Omron CX-Programmer project NewProject (CX-Programmer 9.03)

# PLC APK46: CS1H CPU63
; KARTONIKARKA

## Program TASK_MENAGER (cyclic task 0)
Local symbols
AWARIA_ZBIORCZA 49.15 BOOL  ; AWARIA ZBIORCZA KARTONIKARKI
A_21_22_A1 0.10 BOOL  ; TRIP-NAPĘDÓW
A_21_28 2.04 BOOL  ; ODBLOKOWANIE NAPĘDU GŁÓWNEGO
A_21_A2 0.11 BOOL  ; NAPĘD GŁÓWNY PO BAZOWANIU
A_21_E1 2.05 BOOL  ; JOG-NAPĘDU GŁÓWNEGO
A_21_E2 2.06 BOOL  ; PROGRAM START- TRIP NAPĘDU GŁÓWNEGO
A_21_E3 2.07 BOOL  ; BAZOWANIE NAPĘDU GŁÓWNEGO
A_21_E4 2.08 BOOL  ; INICJACJA NAPĘDU GŁÓWNEGO
A_21_E5 2.09 BOOL  ; input 5 napędu głównego
A_22_28 2.10 BOOL  ; ODBLOKOWANIE NAPĘlDU ZAMYKANIA
A_22_A2 0.12 BOOL  ; NAPĘDU ZAKLEJANIA KARTONIKÓW PO BAZOWANIU
A_22_E1 2.11 BOOL  ; PROGRAM START NAPĘDU ZAMYANA
A_22_E2 2.12 BOOL  ; BAZOWANE NAPĘDU ZAMYKANIA
A_22_E3 2.13 BOOL  ; NCJACJA NAPĘDU ZAMYKANIA
A_22_E4 2.14 BOOL
A_22_E5 2.15 BOOL
CAM_1 25.00 BOOL  ; ZATRZYMANIE SILNIKA
GOT_KART 201.00 BOOL  ; GOTOWOŚĆ KARTONIKARKI DO PRZYJĘCIA PRODUKTU
GOT_KLEJU 0.13 BOOL  ; GOTOWOŚĆ KLEJARKI NORDSON
K_131 2.00 BOOL  ; STYCZNIK-NAPĘD GŁÓWNY
K_132 2.01 BOOL  ; STYCZNIK TRANSPORTER
K_133 2.02 BOOL  ; STYCZNIK KLEJARKA
K_168 3.15 BOOL  ; PRZEKAŻNIK DRUKARKI
K_174 3.11 BOOL  ; PRZEKAŻNIK GOTOWOŚĆ
K_175 3.12 BOOL  ; PRZEKAŻNIK AWARIA
OBW_BEZPIECZ 0.14 BOOL  ; OBWÓD BEZPIECZEŃSTWA
OBW_OSŁON 0.15 BOOL  ; OBWÓD  OSŁON
OBW_STOP 0.14 BOOL  ; OBWÓD STOP
OBW_STOP_OSŁON 0.15 BOOL  ; OBWÓD STOPU I OSŁON
POZ_1024_0 0.00 BOOL  ; BIT 0 ENCODERA
POZ_1024_1 0.01 BOOL  ; BIT 1 ENCODERA
POZ_1024_2 0.02 BOOL  ; BIT 2 ENCODERA
POZ_1024_3 0.03 BOOL  ; BIT 3 ENCODERA
POZ_1024_4 0.04 BOOL  ; BIT 4 ENCODERA
POZ_1024_5 0.05 BOOL  ; BIT 5 ENCODERA
POZ_1024_6 0.06 BOOL  ; BIT 6 ENCODERA
POZ_1024_7 0.07 BOOL  ; BIT 7 ENCODERA
POZ_1024_8 0.08 BOOL  ; BIT 8 ENCODERA
POZ_1024_9 0.09 BOOL  ; BIT 9 ENCODERA
Q_32 1.00 BOOL  ; ZABEZPIECZENIE TERMICZNE TRANSPORTERA
REZERWA_OUT 2.03 BOOL
Restart_specjal_IO A502.00 BOOL
Run_DP 2000.00 BOOL
START W2.00 BOOL  ; ZAŁĄCZONA MASZYNA DO PRACY
S_111L 3.10 BOOL  ; LAMPKA ZAŁĄCZENIE
S_112 1.01 BOOL  ; PRZYCISK ZAŁĄCZENIE
S_113 1.02 BOOL  ; PRZYCISK W YŁĄCZENIE
S_114 1.03 BOOL  ; FOTOKOMÓRKA OBECNOŚCI PAKIETU NA TRANSPORTERZE
S_115 1.04 BOOL  ; OBECNOŚĆ PAKIETU NAD PODNOSZENIEM
S_116 1.05 BOOL  ; FOTOKOMÓRKA OBECNOŚCI KARTONIKA
S_117 1.06 BOOL  ; CZUJNIKI POZYCJI ZAKLEJANIA KARTONIKA
S_118 1.07 BOOL  ; PODNIESIENIE PAKIETU POCZĄTEK
S_121 1.08 BOOL  ; KONIEC SIŁOWNIKA PODNOSZĄCEGO PAKIET
S_122 1.09 BOOL  ; POCZĄTEK SIŁOWNIKA KLAPEK BOCZNYCH
S_123 1.10 BOOL  ; KONIEC SIŁOWNIKA KLAPEK BOCZNYCH
S_124 1.11 BOOL  ; POCZĄTEK SIŁOWNIKA POBIERAJĄCEGO KARTONIK
S_125 1.12 BOOL  ; KONIEC  SIŁOWNIKA POBIERAJĄCEGO KARTONIK
S_126 1.13 BOOL  ; POCZĄTEK SIŁOWNIKA WPYCHAJĄCEGO PAKIET
S_127 1.14 BOOL  ; KONIEC SIŁOWNIKA WPYCHAJĄCEGO
S_128 1.15 BOOL  ; FOTOKOMÓRKA WYJKRYWAJĄCA KARTONIK PRZED SKLEJENIEM
Y_151 3.00 BOOL  ; POBIERANIE KARTONIKÓW
Y_152 3.01 BOOL  ; EŻEKTOR
Y_153 3.02 BOOL  ; PODNOSZENIE PAKIETU
Y_154 3.03 BOOL  ; WPYCHANIE PAKIETU
Y_155 3.04 BOOL  ; KLAPKI BOCZNE
Y_156 3.05 BOOL  ; TRANSPORTER NA STOJAKU
Y_157 3.06 BOOL  ; SPUST POWIETRZA
Y_161 3.08 BOOL  ; ZAWÓR APLIKACJI KLEJU 1
Y_162 3.09 BOOL  ; ZAWÓR APLIKACJI KLEJU 2
ZAŁĄCZ_SILNIKI W0.01 BOOL  ; ZAŁĄCZONE SILNIKI
ZAŁĄCZ_STER W0.00 BOOL  ; ZAŁĄCZONE STEROWANIE
cam_1 25.00 BOOL  ; zatrzymanie napędu głównego
cam_10 25.09 BOOL
cam_2 25.01 BOOL
cam_3 25.02 BOOL
cam_4 25.03 BOOL
cam_5 25.04 BOOL
cam_6 25.05 BOOL
cam_7 25.06 BOOL
cam_8 25.07 BOOL
cam_9 25.08 BOOL

### Section inicjacja

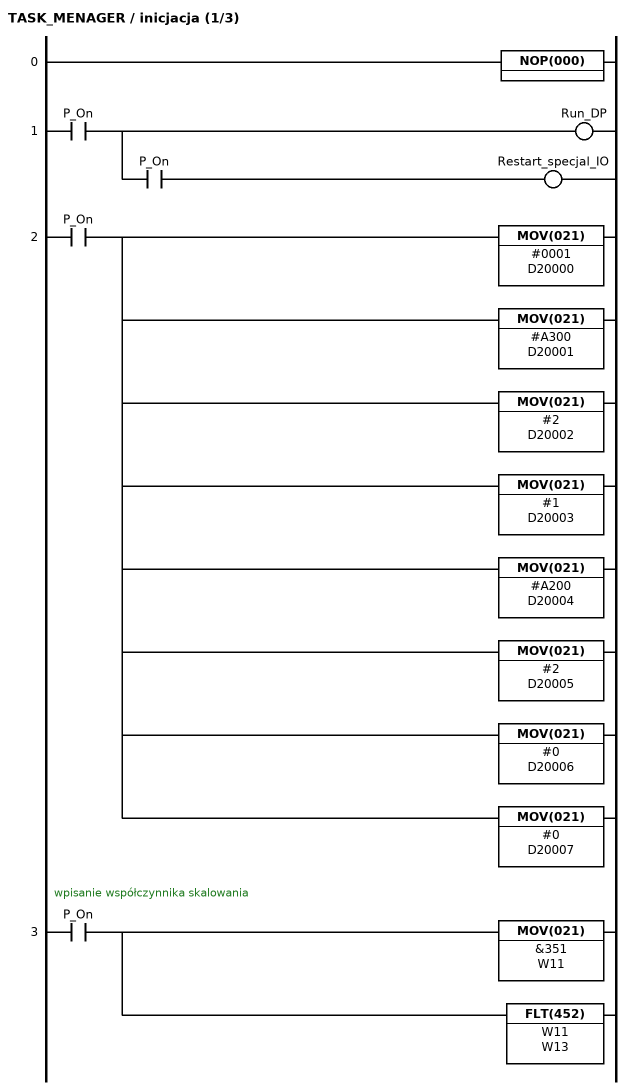
; rung 0
NOP(000)
; rung 1
LD P_On
OUT Run_DP
AND P_On
OUT Restart_specjal_IO
; rung 2
LD P_On
MOV(021) #0001 D20000  // jeden obszar wyjściowy
MOV(021) #A300 D20001  // początek obszaru wyjściowego
MOV(021) #2 D20002  // ustawienie 4 słów wejściowych
MOV(021) #1 D20003  // ustawienie jednego obszaru wyjsciowego
MOV(021) #A200 D20004  // początek obszaru wejściowego
MOV(021) #2 D20005  // ustawienie 4 słów wyjściowych
MOV(021) #0 D20006
MOV(021) #0 D20007
; rung 3: wpisanie współczynnika skalowania
LD P_On
MOV(021) &351 W11
FLT(452) W11 W13

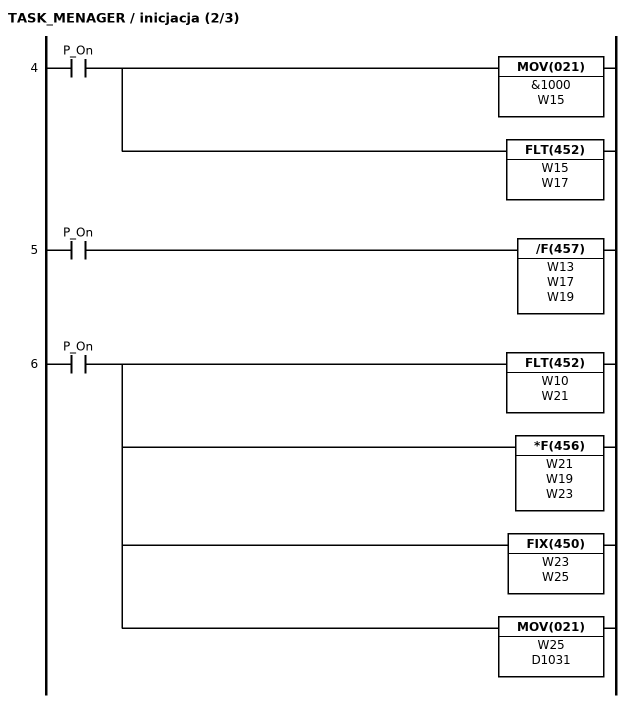
; rung 4
LD P_On
MOV(021) &1000 W15
FLT(452) W15 W17
; rung 5
LD P_On
/F(457) W13 W17 W19  // wspolczynnik 0,351
; rung 6
LD P_On
FLT(452) W10 W21
*F(456) W21 W19 W23
FIX(450) W23 W25
MOV(021) W25 D1031

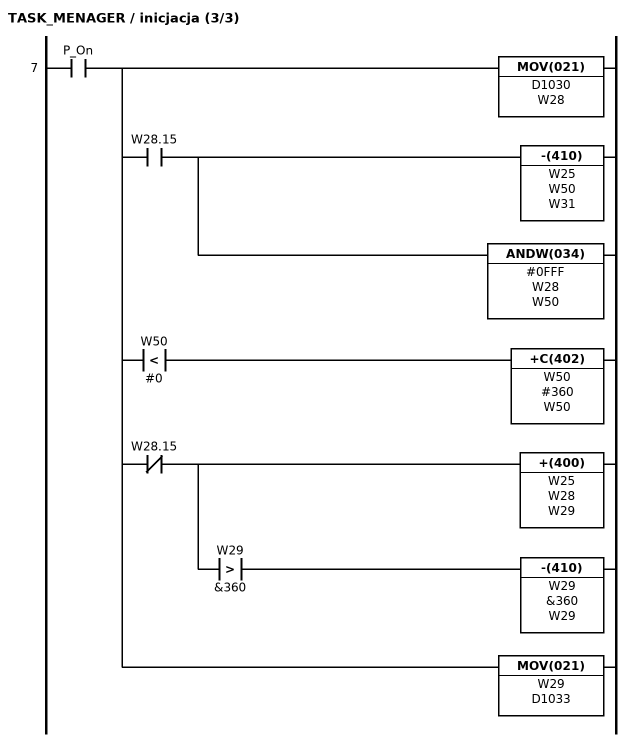
; rung 7
LD P_On
OUT TR0
MOV(021) D1030 W28
AND W28.15
-(410) W25 W50 W31
ANDW(034) #0FFF W28 W50
LD TR0
AND<S(312) W50 #0
+C(402) W50 #360 W50
LD TR0
ANDNOT W28.15
+(400) W25 W28 W29
AND>(320) W29 &360
-(410) W29 &360 W29
LD TR0
MOV(021) W29 D1033

### Section cam_section

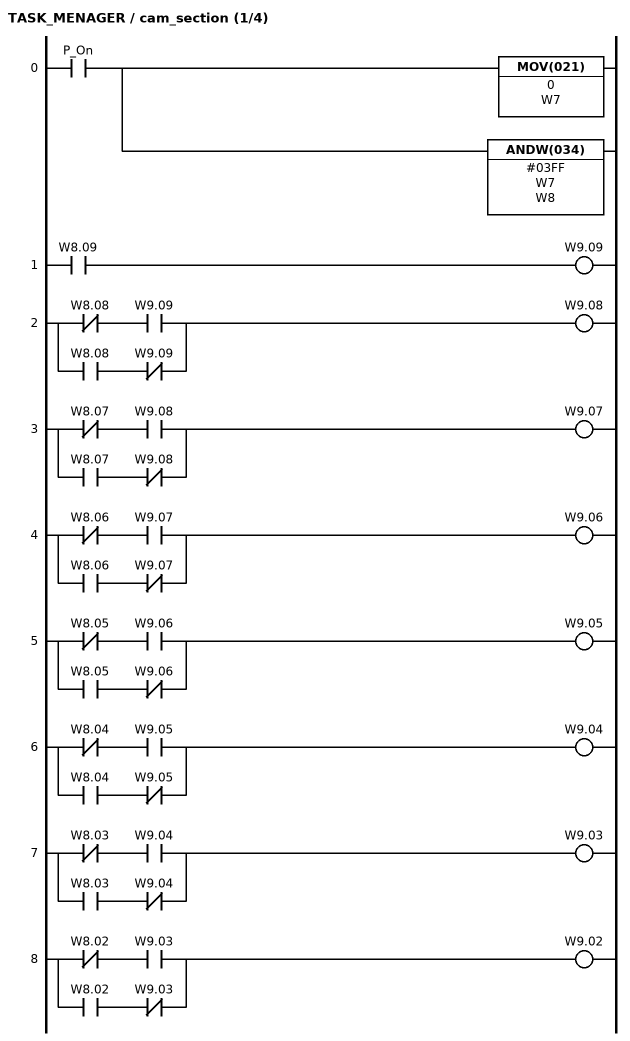
; rung 0
LD P_On
MOV(021) 0 W7
ANDW(034) #03FF W7 W8
; rung 1
LD W8.09
OUT W9.09
; rung 2
LDNOT W8.08
AND W9.09
LD W8.08
ANDNOT W9.09
ORLD
OUT W9.08
; rung 3
LDNOT W8.07
AND W9.08
LD W8.07
ANDNOT W9.08
ORLD
OUT W9.07
; rung 4
LDNOT W8.06
AND W9.07
LD W8.06
ANDNOT W9.07
ORLD
OUT W9.06
; rung 5
LDNOT W8.05
AND W9.06
LD W8.05
ANDNOT W9.06
ORLD
OUT W9.05
; rung 6
LDNOT W8.04
AND W9.05
LD W8.04
ANDNOT W9.05
ORLD
OUT W9.04
; rung 7
LDNOT W8.03
AND W9.04
LD W8.03
ANDNOT W9.04
ORLD
OUT W9.03
; rung 8
LDNOT W8.02
AND W9.03
LD W8.02
ANDNOT W9.03
ORLD
OUT W9.02

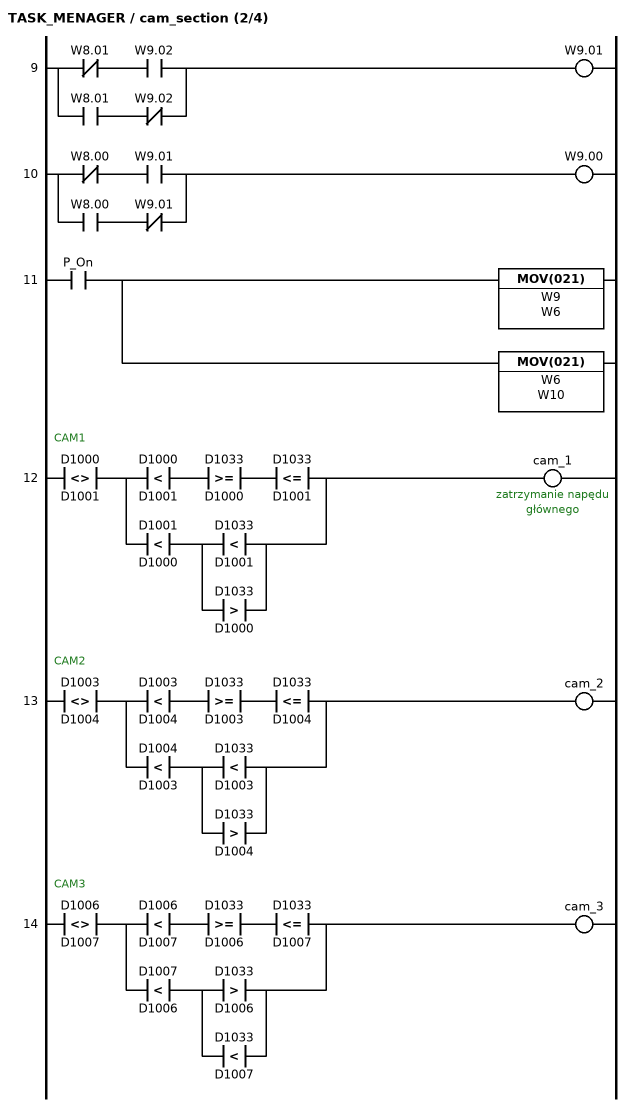
; rung 9
LDNOT W8.01
AND W9.02
LD W8.01
ANDNOT W9.02
ORLD
OUT W9.01
; rung 10
LDNOT W8.00
AND W9.01
LD W8.00
ANDNOT W9.01
ORLD
OUT W9.00
; rung 11
LD P_On
MOV(021) W9 W6
MOV(021) W6 W10
; rung 12: CAM1
LD<>(305) D1000 D1001
LD<(310) D1000 D1001
AND>=(325) D1033 D1000
AND<=(315) D1033 D1001
LD<(310) D1001 D1000
LD<(310) D1033 D1001
OR>(320) D1033 D1000
ANDLD
ORLD
ANDLD
OUT cam_1  ; zatrzymanie napędu głównego
; rung 13: CAM2
LD<>(305) D1003 D1004
LD<(310) D1003 D1004
AND>=(325) D1033 D1003
AND<=(315) D1033 D1004
LD<(310) D1004 D1003
LD<(310) D1033 D1003
OR>(320) D1033 D1004
ANDLD
ORLD
ANDLD
OUT cam_2
; rung 14: CAM3
LD<>(305) D1006 D1007
LD<(310) D1006 D1007
AND>=(325) D1033 D1006
AND<=(315) D1033 D1007
LD<(310) D1007 D1006
LD>(320) D1033 D1006
OR<(310) D1033 D1007
ANDLD
ORLD
ANDLD
OUT cam_3

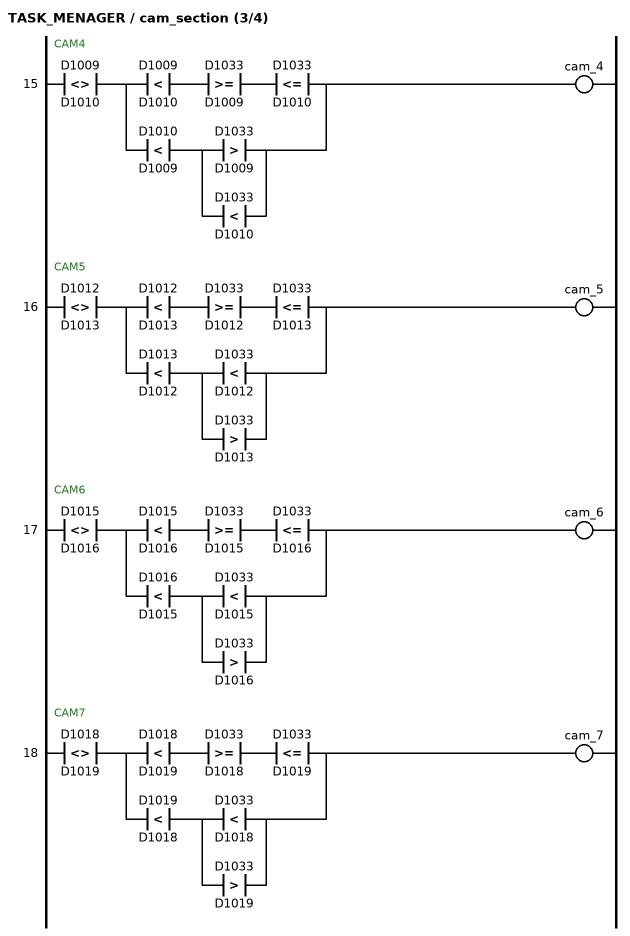
; rung 15: CAM4
LD<>(305) D1009 D1010
LD<(310) D1009 D1010
AND>=(325) D1033 D1009
AND<=(315) D1033 D1010
LD<(310) D1010 D1009
LD>(320) D1033 D1009
OR<(310) D1033 D1010
ANDLD
ORLD
ANDLD
OUT cam_4
; rung 16: CAM5
LD<>(305) D1012 D1013
LD<(310) D1012 D1013
AND>=(325) D1033 D1012
AND<=(315) D1033 D1013
LD<(310) D1013 D1012
LD<(310) D1033 D1012
OR>(320) D1033 D1013
ANDLD
ORLD
ANDLD
OUT cam_5
; rung 17: CAM6
LD<>(305) D1015 D1016
LD<(310) D1015 D1016
AND>=(325) D1033 D1015
AND<=(315) D1033 D1016
LD<(310) D1016 D1015
LD<(310) D1033 D1015
OR>(320) D1033 D1016
ANDLD
ORLD
ANDLD
OUT cam_6
; rung 18: CAM7
LD<>(305) D1018 D1019
LD<(310) D1018 D1019
AND>=(325) D1033 D1018
AND<=(315) D1033 D1019
LD<(310) D1019 D1018
LD<(310) D1033 D1018
OR>(320) D1033 D1019
ANDLD
ORLD
ANDLD
OUT cam_7

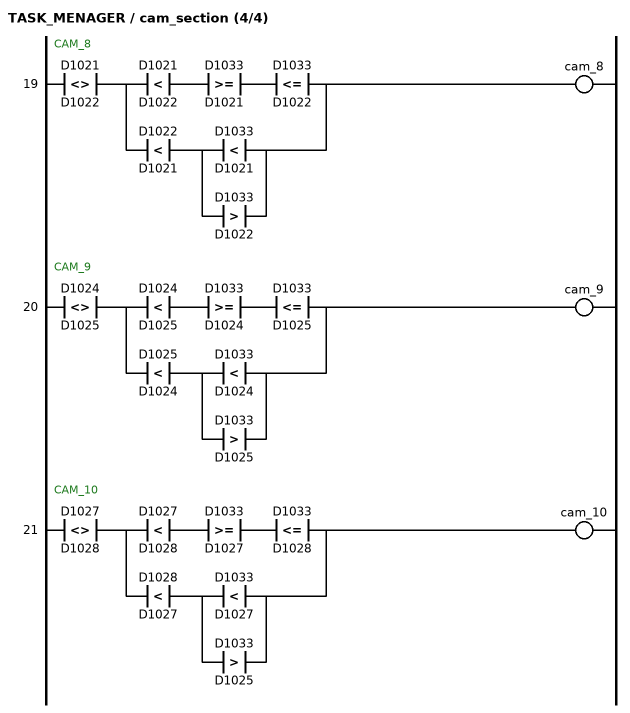
; rung 19: CAM_8
LD<>(305) D1021 D1022
LD<(310) D1021 D1022
AND>=(325) D1033 D1021
AND<=(315) D1033 D1022
LD<(310) D1022 D1021
LD<(310) D1033 D1021
OR>(320) D1033 D1022
ANDLD
ORLD
ANDLD
OUT cam_8
; rung 20: CAM_9
LD<>(305) D1024 D1025
LD<(310) D1024 D1025
AND>=(325) D1033 D1024
AND<=(315) D1033 D1025
LD<(310) D1025 D1024
LD<(310) D1033 D1024
OR>(320) D1033 D1025
ANDLD
ORLD
ANDLD
OUT cam_9
; rung 21: CAM_10
LD<>(305) D1027 D1028
LD<(310) D1027 D1028
AND>=(325) D1033 D1027
AND<=(315) D1033 D1028
LD<(310) D1028 D1027
LD<(310) D1033 D1027
OR>(320) D1033 D1025
ANDLD
ORLD
ANDLD
OUT cam_10

### Section przyjęcie_pakietu

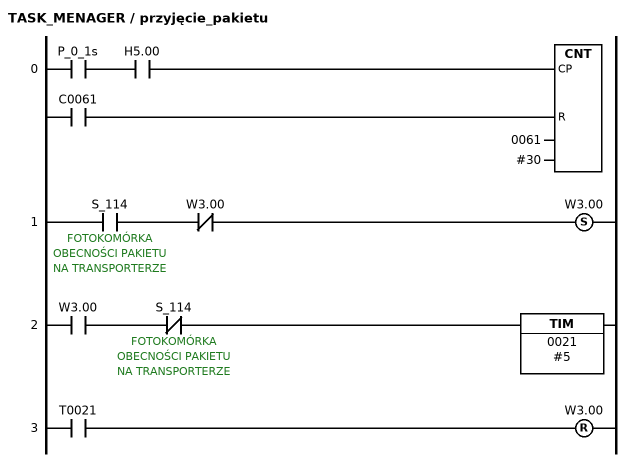
; rung 0
LD P_0_1s
AND H5.00
LD C0061
CNT 0061 #30
; rung 1
LD S_114  ; FOTOKOMÓRKA OBECNOŚCI PAKIETU NA TRANSPORTERZE
ANDNOT W3.00
SET W3.00
; rung 2
LD W3.00
ANDNOT S_114  ; FOTOKOMÓRKA OBECNOŚCI PAKIETU NA TRANSPORTERZE
TIM 0021 #5
; rung 3
LD T0021
RSET W3.00

### Section awaria

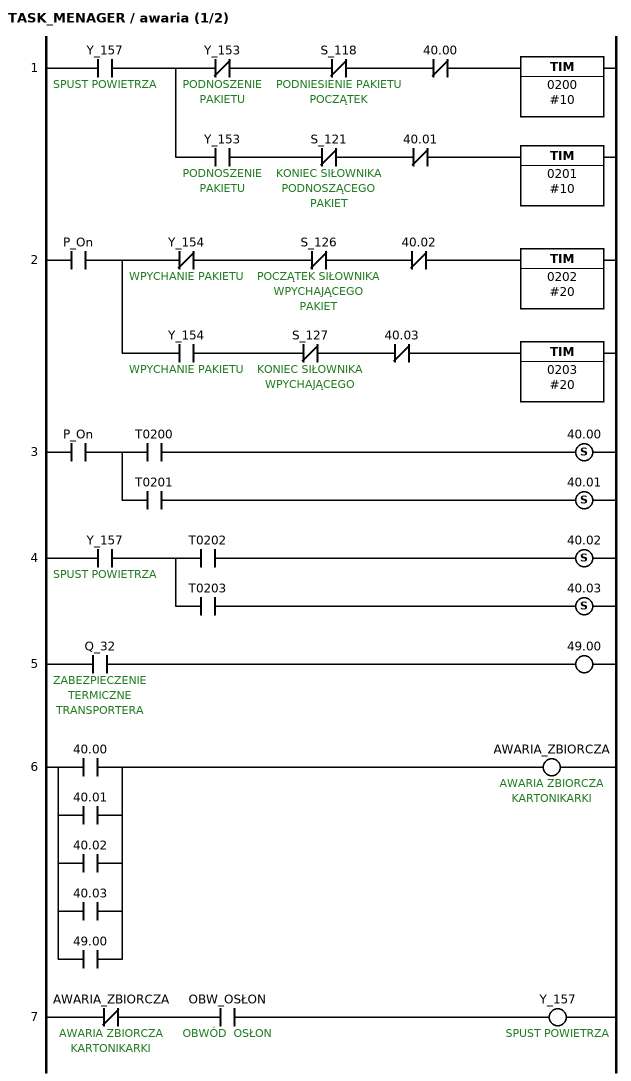
; rung 1
LD Y_157  ; SPUST POWIETRZA
OUT TR0
ANDNOT Y_153  ; PODNOSZENIE PAKIETU
ANDNOT S_118  ; PODNIESIENIE PAKIETU POCZĄTEK
ANDNOT 40.00
TIM 0200 #10
LD TR0
AND Y_153  ; PODNOSZENIE PAKIETU
ANDNOT S_121  ; KONIEC SIŁOWNIKA PODNOSZĄCEGO PAKIET
ANDNOT 40.01
TIM 0201 #10
; rung 2
LD P_On
OUT TR0
ANDNOT Y_154  ; WPYCHANIE PAKIETU
ANDNOT S_126  ; POCZĄTEK SIŁOWNIKA WPYCHAJĄCEGO PAKIET
ANDNOT 40.02
TIM 0202 #20
LD TR0
AND Y_154  ; WPYCHANIE PAKIETU
ANDNOT S_127  ; KONIEC SIŁOWNIKA WPYCHAJĄCEGO
ANDNOT 40.03
TIM 0203 #20
; rung 3
LD P_On
OUT TR0
AND T0200
SET 40.00
LD TR0
AND T0201
SET 40.01
; rung 4
LD Y_157  ; SPUST POWIETRZA
OUT TR0
AND T0202
SET 40.02
LD TR0
AND T0203
SET 40.03
; rung 5
LD Q_32  ; ZABEZPIECZENIE TERMICZNE TRANSPORTERA
OUT 49.00
; rung 6
LD 40.00
OR 40.01
OR 40.02
OR 40.03
OR 49.00
OUT AWARIA_ZBIORCZA  ; AWARIA ZBIORCZA KARTONIKARKI
; rung 7
LDNOT AWARIA_ZBIORCZA  ; AWARIA ZBIORCZA KARTONIKARKI
AND OBW_OSŁON  ; OBWÓD  OSŁON
OUT Y_157  ; SPUST POWIETRZA

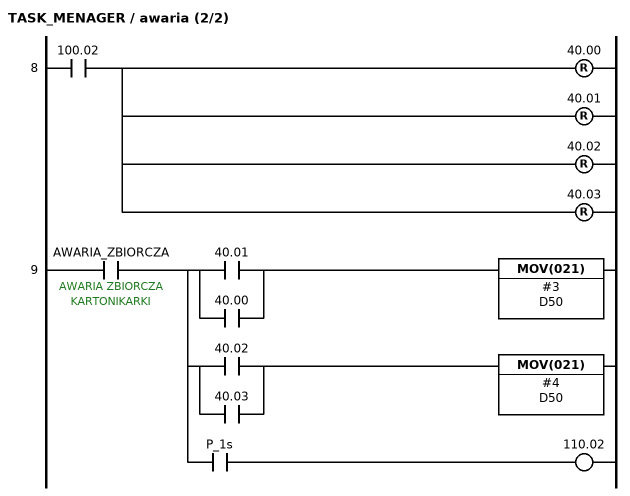
; rung 8
LD 100.02
RSET 40.00
RSET 40.01
RSET 40.02
RSET 40.03
; rung 9
LD AWARIA_ZBIORCZA  ; AWARIA ZBIORCZA KARTONIKARKI
OUT TR0
LD 40.01
OR 40.00
ANDLD
MOV(021) #3 D50
LD TR0
LD 40.02
OR 40.03
ANDLD
MOV(021) #4 D50
LD TR0
AND P_1s
OUT 110.02

### Section gotowość

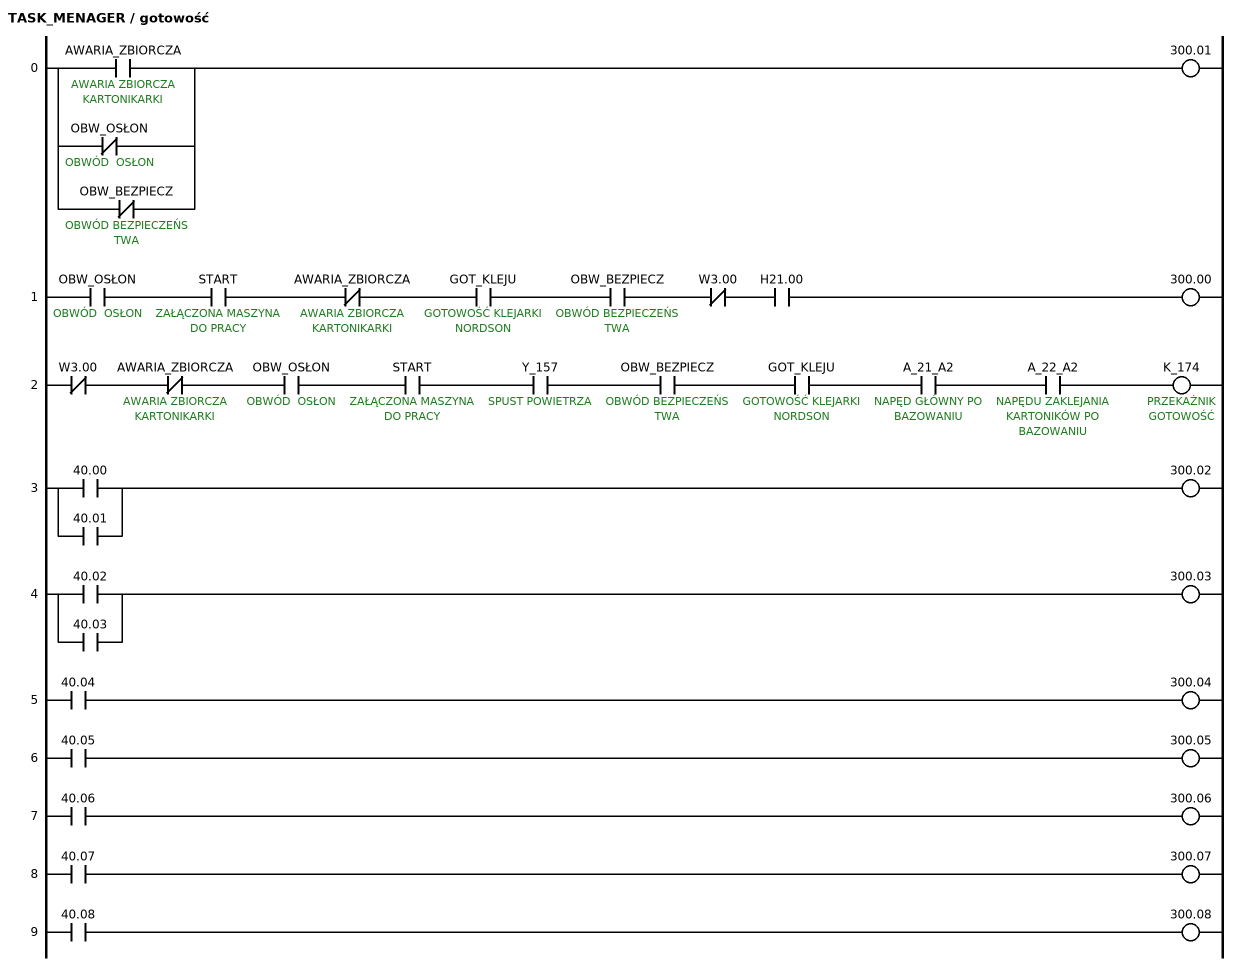
; rung 0
LD AWARIA_ZBIORCZA  ; AWARIA ZBIORCZA KARTONIKARKI
ORNOT OBW_OSŁON  ; OBWÓD  OSŁON
ORNOT OBW_BEZPIECZ  ; OBWÓD BEZPIECZEŃSTWA
OUT 300.01
; rung 1
LD OBW_OSŁON  ; OBWÓD  OSŁON
AND START  ; ZAŁĄCZONA MASZYNA DO PRACY
ANDNOT AWARIA_ZBIORCZA  ; AWARIA ZBIORCZA KARTONIKARKI
AND GOT_KLEJU  ; GOTOWOŚĆ KLEJARKI NORDSON
AND OBW_BEZPIECZ  ; OBWÓD BEZPIECZEŃSTWA
ANDNOT W3.00
AND H21.00
OUT 300.00
; rung 2
LDNOT W3.00
ANDNOT AWARIA_ZBIORCZA  ; AWARIA ZBIORCZA KARTONIKARKI
AND OBW_OSŁON  ; OBWÓD  OSŁON
AND START  ; ZAŁĄCZONA MASZYNA DO PRACY
AND Y_157  ; SPUST POWIETRZA
AND OBW_BEZPIECZ  ; OBWÓD BEZPIECZEŃSTWA
AND GOT_KLEJU  ; GOTOWOŚĆ KLEJARKI NORDSON
AND A_21_A2  ; NAPĘD GŁÓWNY PO BAZOWANIU
AND A_22_A2  ; NAPĘDU ZAKLEJANIA KARTONIKÓW PO BAZOWANIU
OUT K_174  ; PRZEKAŻNIK GOTOWOŚĆ
; rung 3
LD 40.00
OR 40.01
OUT 300.02
; rung 4
LD 40.02
OR 40.03
OUT 300.03
; rung 5
LD 40.04
OUT 300.04
; rung 6
LD 40.05
OUT 300.05
; rung 7
LD 40.06
OUT 300.06
; rung 8
LD 40.07
OUT 300.07
; rung 9
LD 40.08
OUT 300.08

### Section podniesienie_pakietu

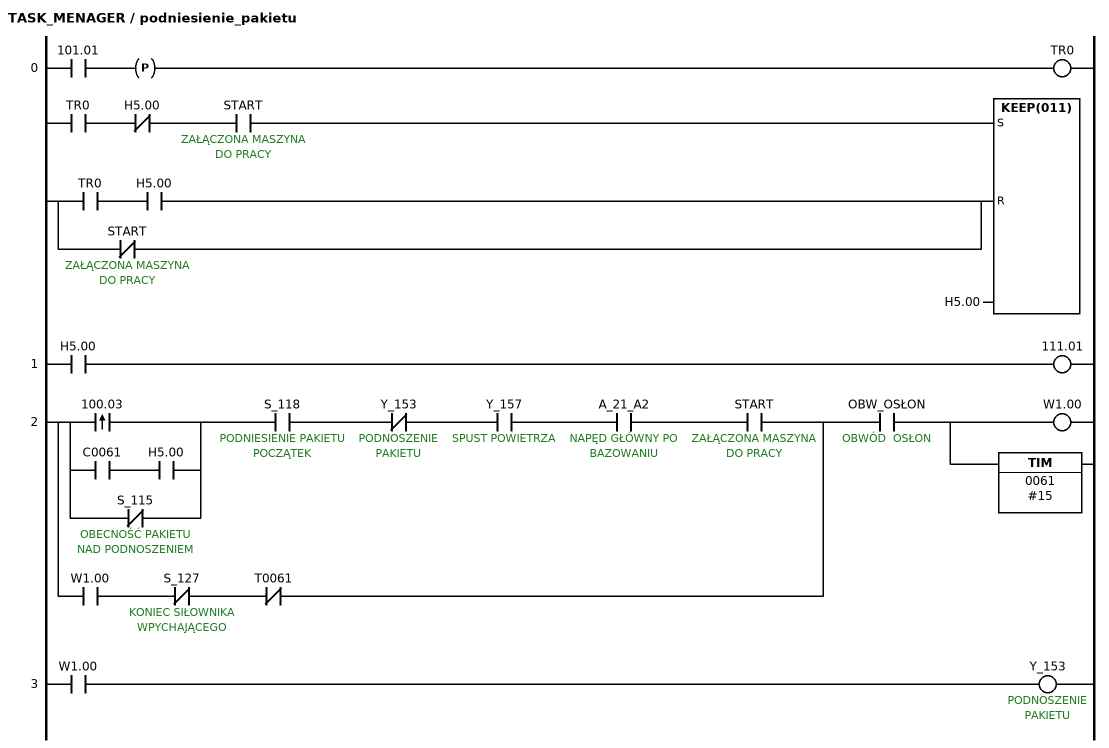
; rung 0
LD 101.01
UP(521)
OUT TR0
ANDNOT H5.00
AND START  ; ZAŁĄCZONA MASZYNA DO PRACY
LD TR0
AND H5.00
ORNOT START  ; ZAŁĄCZONA MASZYNA DO PRACY
KEEP(011) H5.00
; rung 1
LD H5.00
OUT 111.01
; rung 2
@LD 100.03
LD C0061
AND H5.00
ORLD
ORNOT S_115  ; OBECNOŚĆ PAKIETU NAD PODNOSZENIEM
AND S_118  ; PODNIESIENIE PAKIETU POCZĄTEK
ANDNOT Y_153  ; PODNOSZENIE PAKIETU
AND Y_157  ; SPUST POWIETRZA
AND A_21_A2  ; NAPĘD GŁÓWNY PO BAZOWANIU
AND START  ; ZAŁĄCZONA MASZYNA DO PRACY
LD W1.00
ANDNOT S_127  ; KONIEC SIŁOWNIKA WPYCHAJĄCEGO
ANDNOT T0061
ORLD
AND OBW_OSŁON  ; OBWÓD  OSŁON
OUT W1.00
TIM 0061 #15
; rung 3
LD W1.00
OUT Y_153  ; PODNOSZENIE PAKIETU

### Section wepchnięcie_pakietu

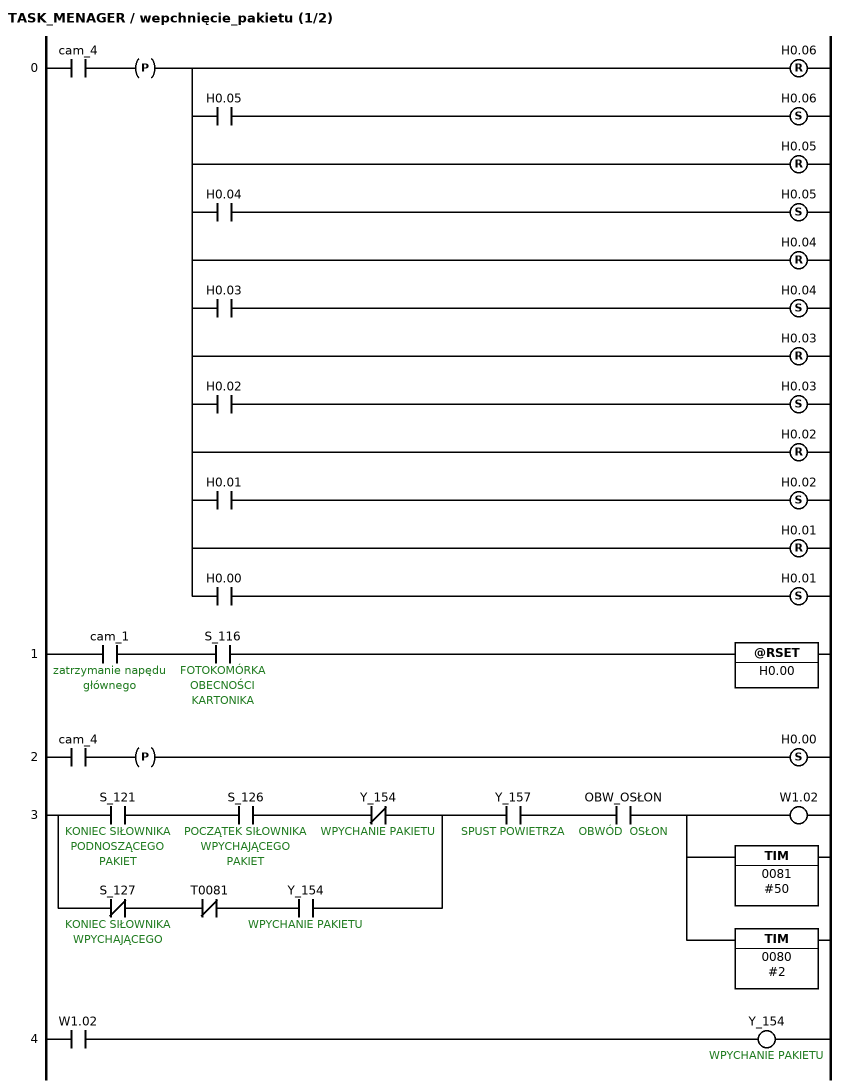
; rung 0
LD cam_4
UP(521)
OUT TR0
RSET H0.06
AND H0.05
SET H0.06
LD TR0
RSET H0.05
AND H0.04
SET H0.05
LD TR0
RSET H0.04
AND H0.03
SET H0.04
LD TR0
RSET H0.03
AND H0.02
SET H0.03
LD TR0
RSET H0.02
AND H0.01
SET H0.02
LD TR0
RSET H0.01
AND H0.00
SET H0.01
; rung 1
LD cam_1  ; zatrzymanie napędu głównego
AND S_116  ; FOTOKOMÓRKA OBECNOŚCI KARTONIKA
@RSET H0.00
; rung 2
LD cam_4
UP(521)
SET H0.00
; rung 3
LD S_121  ; KONIEC SIŁOWNIKA PODNOSZĄCEGO PAKIET
AND S_126  ; POCZĄTEK SIŁOWNIKA WPYCHAJĄCEGO PAKIET
ANDNOT Y_154  ; WPYCHANIE PAKIETU
LDNOT S_127  ; KONIEC SIŁOWNIKA WPYCHAJĄCEGO
ANDNOT T0081
AND Y_154  ; WPYCHANIE PAKIETU
ORLD
AND Y_157  ; SPUST POWIETRZA
AND OBW_OSŁON  ; OBWÓD  OSŁON
OUT W1.02
TIM 0081 #50
TIM 0080 #2
; rung 4
LD W1.02
OUT Y_154  ; WPYCHANIE PAKIETU

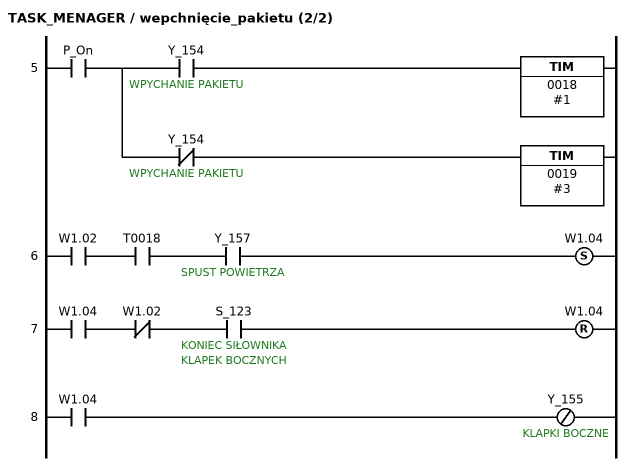
; rung 5
LD P_On
OUT TR0
AND Y_154  ; WPYCHANIE PAKIETU
TIM 0018 #1
LD TR0
ANDNOT Y_154  ; WPYCHANIE PAKIETU
TIM 0019 #3
; rung 6
LD W1.02
AND T0018
AND Y_157  ; SPUST POWIETRZA
SET W1.04
; rung 7
LD W1.04
ANDNOT W1.02
AND S_123  ; KONIEC SIŁOWNIKA KLAPEK BOCZNYCH
RSET W1.04
; rung 8
LD W1.04
OUTNOT Y_155  ; KLAPKI BOCZNE

### Section napęd_główny

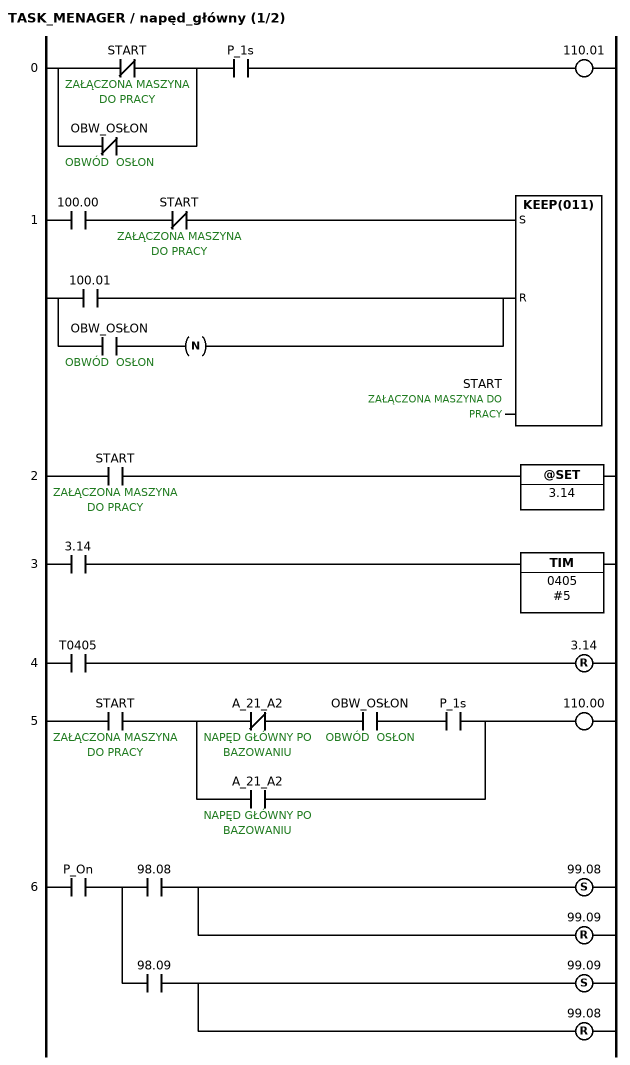
; rung 0
LDNOT START  ; ZAŁĄCZONA MASZYNA DO PRACY
ORNOT OBW_OSŁON  ; OBWÓD  OSŁON
AND P_1s
OUT 110.01
; rung 1
LD 100.00
ANDNOT START  ; ZAŁĄCZONA MASZYNA DO PRACY
LD 100.01
LD OBW_OSŁON  ; OBWÓD  OSŁON
DOWN(522)
ORLD
KEEP(011) START  ; ZAŁĄCZONA MASZYNA DO PRACY
; rung 2
LD START  ; ZAŁĄCZONA MASZYNA DO PRACY
@SET 3.14
; rung 3
LD 3.14
TIM 0405 #5
; rung 4
LD T0405
RSET 3.14
; rung 5
LD START  ; ZAŁĄCZONA MASZYNA DO PRACY
LDNOT A_21_A2  ; NAPĘD GŁÓWNY PO BAZOWANIU
AND OBW_OSŁON  ; OBWÓD  OSŁON
AND P_1s
OR A_21_A2  ; NAPĘD GŁÓWNY PO BAZOWANIU
ANDLD
OUT 110.00
; rung 6
LD P_On
OUT TR0
AND 98.08
SET 99.08
RSET 99.09
LD TR0
AND 98.09
SET 99.09
RSET 99.08

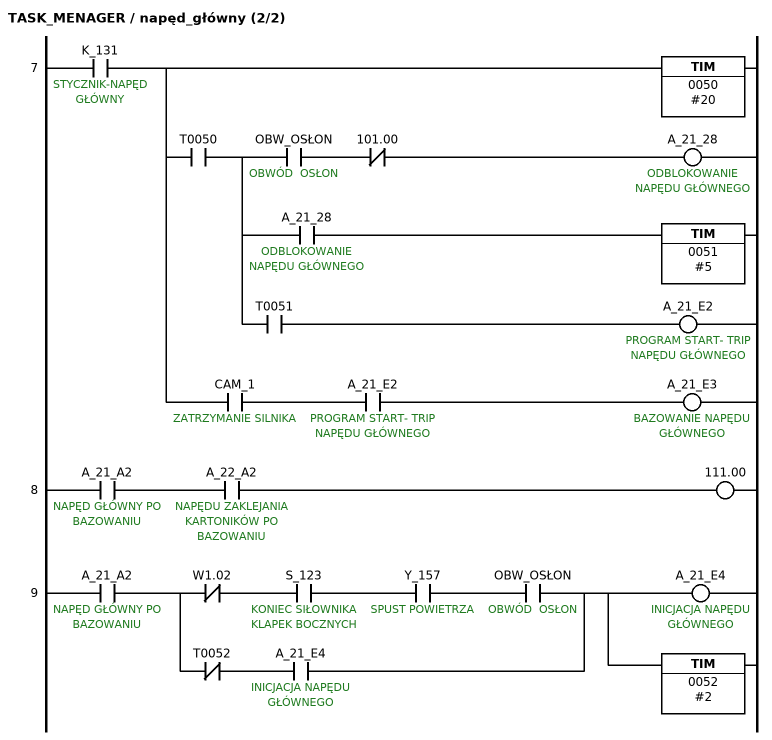
; rung 7
LD K_131  ; STYCZNIK-NAPĘD GŁÓWNY
OUT TR0
TIM 0050 #20
AND T0050
OUT TR1
AND OBW_OSŁON  ; OBWÓD  OSŁON
ANDNOT 101.00
OUT A_21_28  ; ODBLOKOWANIE NAPĘDU GŁÓWNEGO
LD TR1
AND A_21_28  ; ODBLOKOWANIE NAPĘDU GŁÓWNEGO
TIM 0051 #5
LD TR1
AND T0051
OUT A_21_E2  ; PROGRAM START- TRIP NAPĘDU GŁÓWNEGO
LD TR0
AND CAM_1  ; ZATRZYMANIE SILNIKA
AND A_21_E2  ; PROGRAM START- TRIP NAPĘDU GŁÓWNEGO
OUT A_21_E3  ; BAZOWANIE NAPĘDU GŁÓWNEGO
; rung 8
LD A_21_A2  ; NAPĘD GŁÓWNY PO BAZOWANIU
AND A_22_A2  ; NAPĘDU ZAKLEJANIA KARTONIKÓW PO BAZOWANIU
OUT 111.00
; rung 9
LD A_21_A2  ; NAPĘD GŁÓWNY PO BAZOWANIU
LDNOT W1.02
AND S_123  ; KONIEC SIŁOWNIKA KLAPEK BOCZNYCH
AND Y_157  ; SPUST POWIETRZA
AND OBW_OSŁON  ; OBWÓD  OSŁON
LDNOT T0052
AND A_21_E4  ; INICJACJA NAPĘDU GŁÓWNEGO
ORLD
ANDLD
OUT A_21_E4  ; INICJACJA NAPĘDU GŁÓWNEGO
TIM 0052 #2

### Section napęd_zamykania

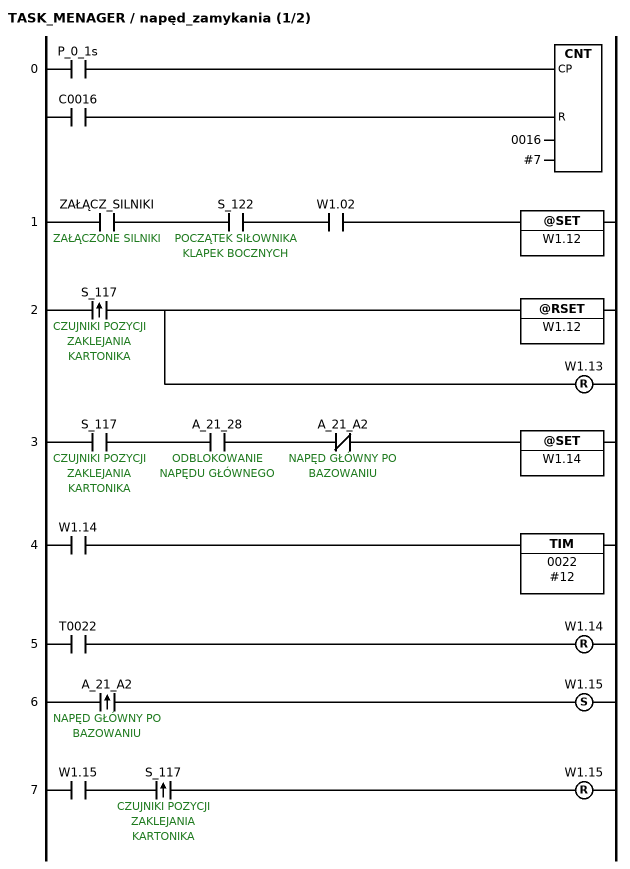
; rung 0
LD P_0_1s
LD C0016
CNT 0016 #7
; rung 1
LD ZAŁĄCZ_SILNIKI  ; ZAŁĄCZONE SILNIKI
AND S_122  ; POCZĄTEK SIŁOWNIKA KLAPEK BOCZNYCH
AND W1.02
@SET W1.12
; rung 2
@LD S_117  ; CZUJNIKI POZYCJI ZAKLEJANIA KARTONIKA
@RSET W1.12
RSET W1.13
; rung 3
LD S_117  ; CZUJNIKI POZYCJI ZAKLEJANIA KARTONIKA
AND A_21_28  ; ODBLOKOWANIE NAPĘDU GŁÓWNEGO
ANDNOT A_21_A2  ; NAPĘD GŁÓWNY PO BAZOWANIU
@SET W1.14
; rung 4
LD W1.14
TIM 0022 #12
; rung 5
LD T0022
RSET W1.14
; rung 6
@LD A_21_A2  ; NAPĘD GŁÓWNY PO BAZOWANIU
SET W1.15
; rung 7
LD W1.15
@AND S_117  ; CZUJNIKI POZYCJI ZAKLEJANIA KARTONIKA
RSET W1.15

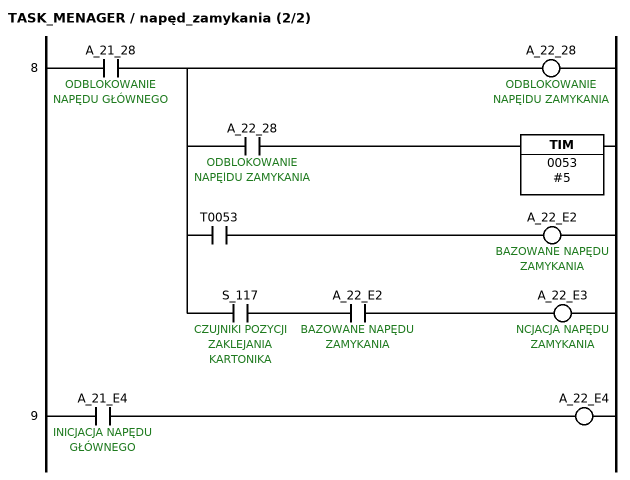
; rung 8
LD A_21_28  ; ODBLOKOWANIE NAPĘDU GŁÓWNEGO
OUT TR0
OUT A_22_28  ; ODBLOKOWANIE NAPĘlDU ZAMYKANIA
AND A_22_28  ; ODBLOKOWANIE NAPĘlDU ZAMYKANIA
TIM 0053 #5
LD TR0
AND T0053
OUT A_22_E2  ; BAZOWANE NAPĘDU ZAMYKANIA
LD TR0
AND S_117  ; CZUJNIKI POZYCJI ZAKLEJANIA KARTONIKA
AND A_22_E2  ; BAZOWANE NAPĘDU ZAMYKANIA
OUT A_22_E3  ; NCJACJA NAPĘDU ZAMYKANIA
; rung 9
LD A_21_E4  ; INICJACJA NAPĘDU GŁÓWNEGO
OUT A_22_E4

### Section pobieranie_kartonika

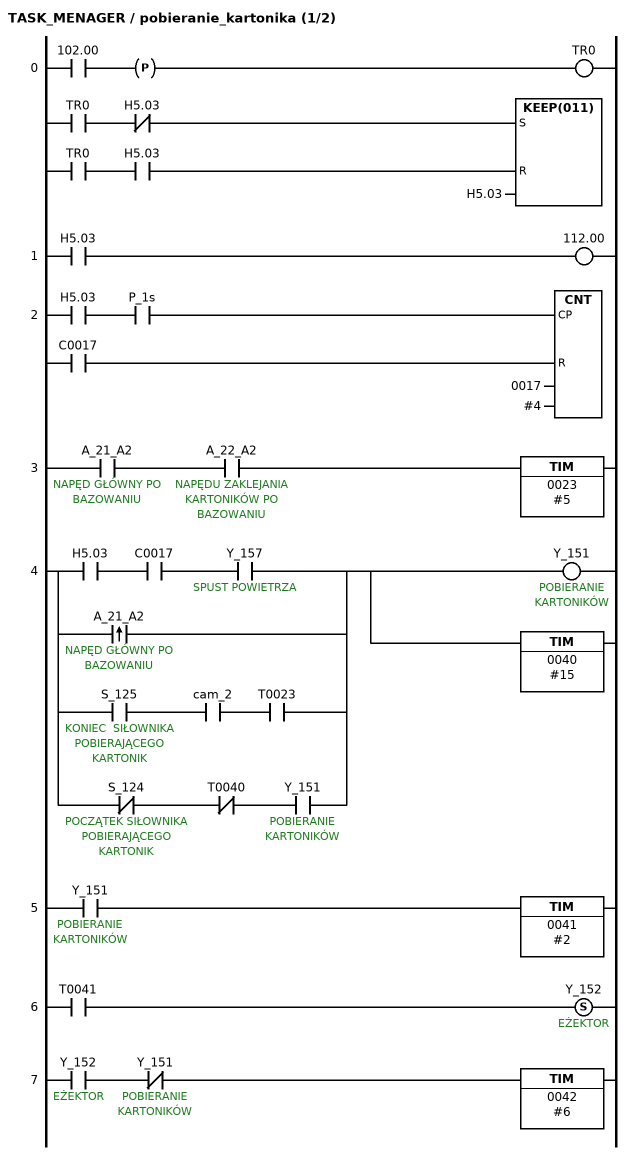
; rung 0
LD 102.00
UP(521)
OUT TR0
ANDNOT H5.03
LD TR0
AND H5.03
KEEP(011) H5.03
; rung 1
LD H5.03
OUT 112.00
; rung 2
LD H5.03
AND P_1s
LD C0017
CNT 0017 #4
; rung 3
LD A_21_A2  ; NAPĘD GŁÓWNY PO BAZOWANIU
AND A_22_A2  ; NAPĘDU ZAKLEJANIA KARTONIKÓW PO BAZOWANIU
TIM 0023 #5
; rung 4
LD H5.03
AND C0017
AND Y_157  ; SPUST POWIETRZA
@OR A_21_A2  ; NAPĘD GŁÓWNY PO BAZOWANIU
LD S_125  ; KONIEC  SIŁOWNIKA POBIERAJĄCEGO KARTONIK
AND cam_2
AND T0023
ORLD
LDNOT S_124  ; POCZĄTEK SIŁOWNIKA POBIERAJĄCEGO KARTONIK
ANDNOT T0040
AND Y_151  ; POBIERANIE KARTONIKÓW
ORLD
OUT Y_151  ; POBIERANIE KARTONIKÓW
TIM 0040 #15
; rung 5
LD Y_151  ; POBIERANIE KARTONIKÓW
TIM 0041 #2
; rung 6
LD T0041
SET Y_152  ; EŻEKTOR
; rung 7
LD Y_152  ; EŻEKTOR
ANDNOT Y_151  ; POBIERANIE KARTONIKÓW
TIM 0042 #6

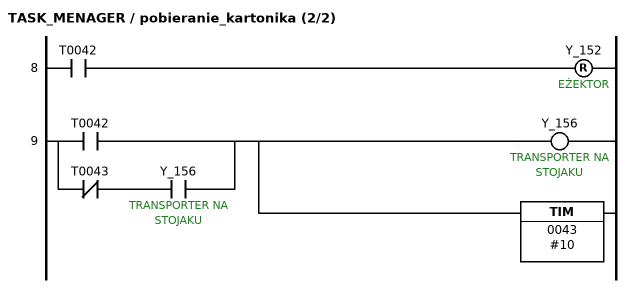
; rung 8
LD T0042
RSET Y_152  ; EŻEKTOR
; rung 9
LD T0042
LDNOT T0043
AND Y_156  ; TRANSPORTER NA STOJAKU
ORLD
OUT Y_156  ; TRANSPORTER NA STOJAKU
TIM 0043 #10

### Section klejenie_kartonika

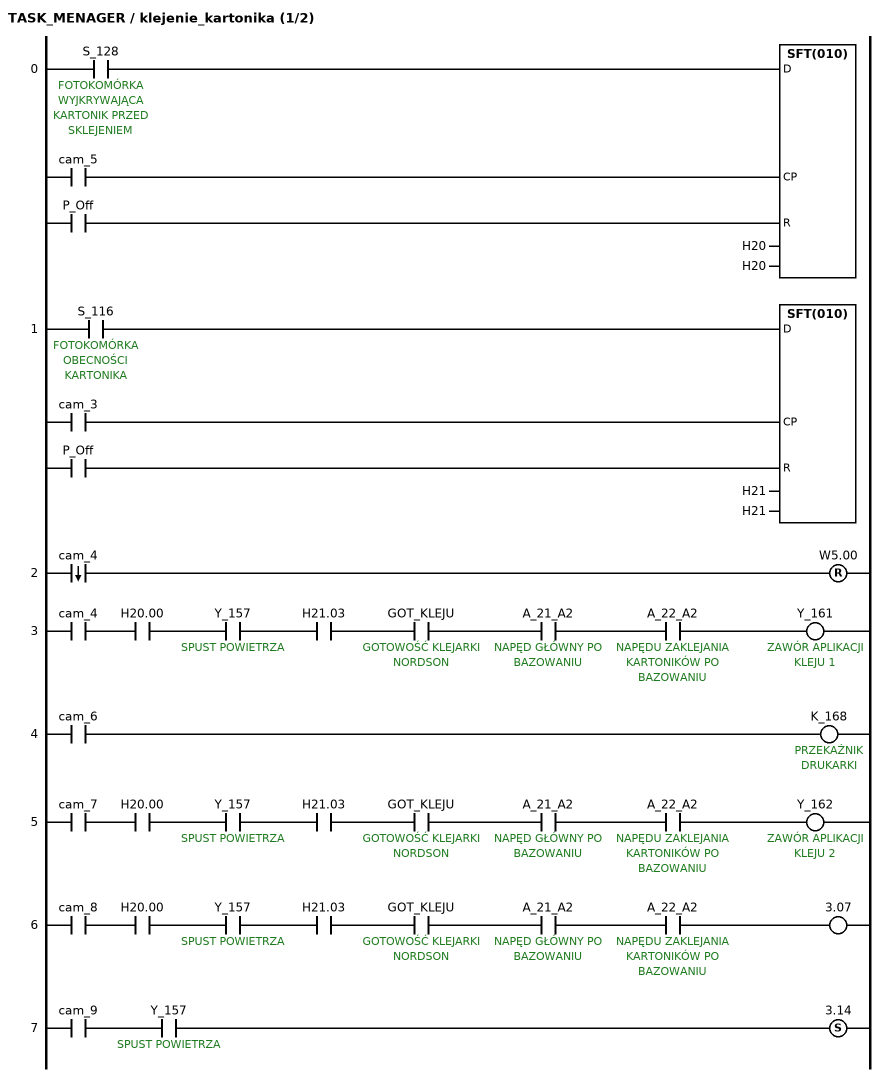
; rung 0
LD S_128  ; FOTOKOMÓRKA WYJKRYWAJĄCA KARTONIK PRZED SKLEJENIEM
LD cam_5
LD P_Off
SFT(010) H20 H20
; rung 1
LD S_116  ; FOTOKOMÓRKA OBECNOŚCI KARTONIKA
LD cam_3
LD P_Off
SFT(010) H21 H21
; rung 2
%LD cam_4
RSET W5.00
; rung 3
LD cam_4
AND H20.00
AND Y_157  ; SPUST POWIETRZA
AND H21.03
AND GOT_KLEJU  ; GOTOWOŚĆ KLEJARKI NORDSON
AND A_21_A2  ; NAPĘD GŁÓWNY PO BAZOWANIU
AND A_22_A2  ; NAPĘDU ZAKLEJANIA KARTONIKÓW PO BAZOWANIU
OUT Y_161  ; ZAWÓR APLIKACJI KLEJU 1
; rung 4
LD cam_6
OUT K_168  ; PRZEKAŻNIK DRUKARKI
; rung 5
LD cam_7
AND H20.00
AND Y_157  ; SPUST POWIETRZA
AND H21.03
AND GOT_KLEJU  ; GOTOWOŚĆ KLEJARKI NORDSON
AND A_21_A2  ; NAPĘD GŁÓWNY PO BAZOWANIU
AND A_22_A2  ; NAPĘDU ZAKLEJANIA KARTONIKÓW PO BAZOWANIU
OUT Y_162  ; ZAWÓR APLIKACJI KLEJU 2
; rung 6
LD cam_8
AND H20.00
AND Y_157  ; SPUST POWIETRZA
AND H21.03
AND GOT_KLEJU  ; GOTOWOŚĆ KLEJARKI NORDSON
AND A_21_A2  ; NAPĘD GŁÓWNY PO BAZOWANIU
AND A_22_A2  ; NAPĘDU ZAKLEJANIA KARTONIKÓW PO BAZOWANIU
OUT 3.07
; rung 7
LD cam_9
AND Y_157  ; SPUST POWIETRZA
SET 3.14

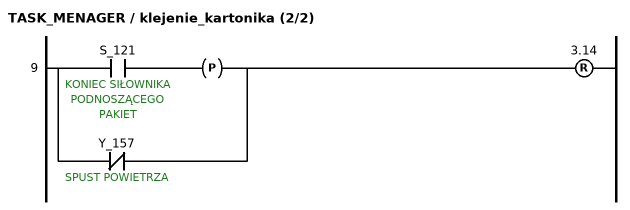
; rung 9
LD S_121  ; KONIEC SIŁOWNIKA PODNOSZĄCEGO PAKIET
UP(521)
ORNOT Y_157  ; SPUST POWIETRZA
RSET 3.14

### Section załączenie

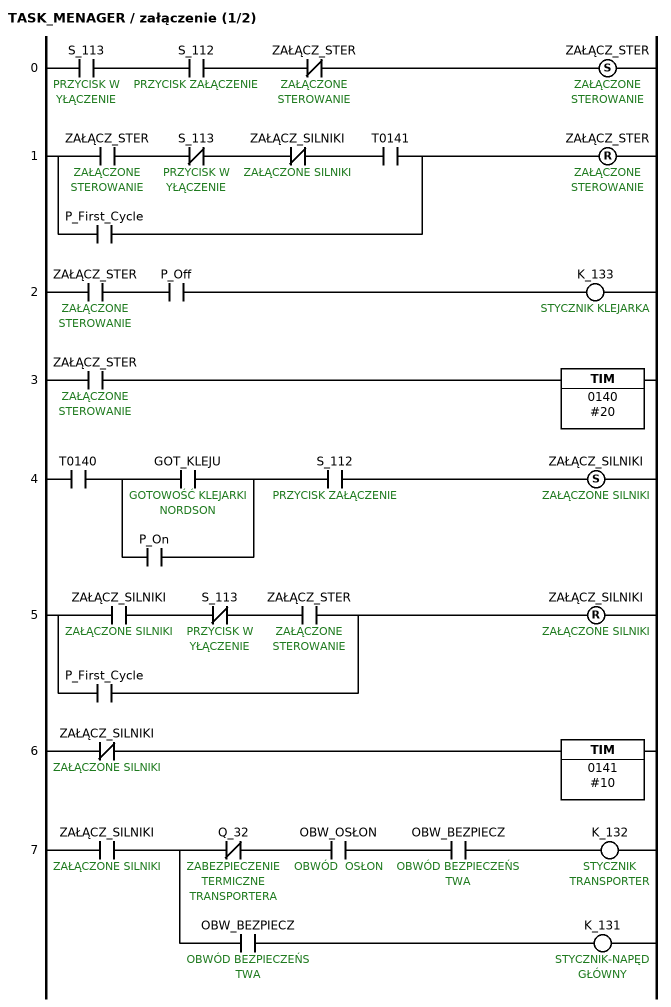
; rung 0
LD S_113  ; PRZYCISK W YŁĄCZENIE
AND S_112  ; PRZYCISK ZAŁĄCZENIE
ANDNOT ZAŁĄCZ_STER  ; ZAŁĄCZONE STEROWANIE
SET ZAŁĄCZ_STER  ; ZAŁĄCZONE STEROWANIE
; rung 1
LD ZAŁĄCZ_STER  ; ZAŁĄCZONE STEROWANIE
ANDNOT S_113  ; PRZYCISK W YŁĄCZENIE
ANDNOT ZAŁĄCZ_SILNIKI  ; ZAŁĄCZONE SILNIKI
AND T0141
OR P_First_Cycle
RSET ZAŁĄCZ_STER  ; ZAŁĄCZONE STEROWANIE
; rung 2
LD ZAŁĄCZ_STER  ; ZAŁĄCZONE STEROWANIE
AND P_Off
OUT K_133  ; STYCZNIK KLEJARKA
; rung 3
LD ZAŁĄCZ_STER  ; ZAŁĄCZONE STEROWANIE
TIM 0140 #20
; rung 4
LD T0140
LD GOT_KLEJU  ; GOTOWOŚĆ KLEJARKI NORDSON
OR P_On
ANDLD
AND S_112  ; PRZYCISK ZAŁĄCZENIE
SET ZAŁĄCZ_SILNIKI  ; ZAŁĄCZONE SILNIKI
; rung 5
LD ZAŁĄCZ_SILNIKI  ; ZAŁĄCZONE SILNIKI
ANDNOT S_113  ; PRZYCISK W YŁĄCZENIE
AND ZAŁĄCZ_STER  ; ZAŁĄCZONE STEROWANIE
OR P_First_Cycle
RSET ZAŁĄCZ_SILNIKI  ; ZAŁĄCZONE SILNIKI
; rung 6
LDNOT ZAŁĄCZ_SILNIKI  ; ZAŁĄCZONE SILNIKI
TIM 0141 #10
; rung 7
LD ZAŁĄCZ_SILNIKI  ; ZAŁĄCZONE SILNIKI
OUT TR0
ANDNOT Q_32  ; ZABEZPIECZENIE TERMICZNE TRANSPORTERA
AND OBW_OSŁON  ; OBWÓD  OSŁON
AND OBW_BEZPIECZ  ; OBWÓD BEZPIECZEŃSTWA
OUT K_132  ; STYCZNIK TRANSPORTER
LD TR0
AND OBW_BEZPIECZ  ; OBWÓD BEZPIECZEŃSTWA
OUT K_131  ; STYCZNIK-NAPĘD GŁÓWNY

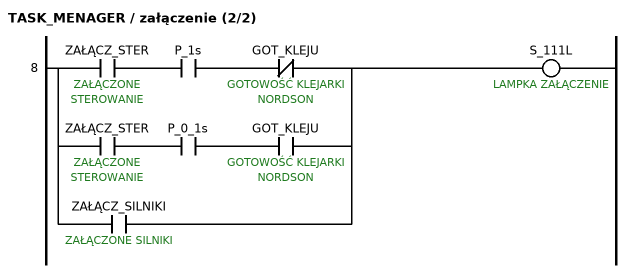
; rung 8
LD ZAŁĄCZ_STER  ; ZAŁĄCZONE STEROWANIE
AND P_1s
ANDNOT GOT_KLEJU  ; GOTOWOŚĆ KLEJARKI NORDSON
LD ZAŁĄCZ_STER  ; ZAŁĄCZONE STEROWANIE
AND P_0_1s
AND GOT_KLEJU  ; GOTOWOŚĆ KLEJARKI NORDSON
ORLD
OR ZAŁĄCZ_SILNIKI  ; ZAŁĄCZONE SILNIKI
OUT S_111L  ; LAMPKA ZAŁĄCZENIE

### Section statystyka

